// TIA Portal V20 export
// export: Created 2026-07-10T11:12:29.0471858Z, ExportSetting WithDefaults, DisplayName Totally Integrated Automation Portal, DisplayVersion V20, DisplayName TIA Portal Openness, DisplayVersion V20, DisplayName TIA Portal Version Control Interface, DisplayVersion V20, DisplayName STEP 7 Professional, DisplayVersion V20, DisplayName STEP 7 Safety, DisplayVersion V20, DisplayName WinCC Basic/Comfort/Advanced, DisplayVersion V20, DisplayName WinCC Unified, DisplayVersion V20
DATA_BLOCK "ChlorMode_DB"   // DB6
VERSION : 0.1
// stored: AutoNumber true, DBAccessibleFromOPCUA true, InstanceOfName ChlorMode, InstanceOfType FB
"ChlorMode"
   // VAR
   //    WaterLevel : Real;
   //    WaterPulse_RT { S7_SetPoint := 'True'} : R_TRIG;
   //    PulseSetpoint { S7_SetPoint := 'True'} : Real;
   //    FreqTON { S7_SetPoint := 'True'} : TON_TIME;
   //    LevelAlarm { S7_SetPoint := 'True'} : Bool;
   //    DelayTOF { S7_SetPoint := 'True'} : TOF_TIME;
   //    PulseGen { S7_SetPoint := 'True'} : TP_TIME;
   //    DoserValue { S7_SetPoint := 'True'} : Real;
   //    DoserPreValue : Real;
   //    StopTrig { S7_SetPoint := 'True'} : R_TRIG;
   //    StartTrig { S7_SetPoint := 'True'} : R_TRIG;
   //    ChlorMeasurment { S7_SetPoint := 'True'} : "ChlorMeasurment";
   //    BlockDosing { S7_SetPoint := 'True'} : Bool;
   //    EnableMeasureTime : Real;
   //    BlockDosingTime : Real;
   // END_VAR
BEGIN
END_DATA_BLOCK
